(* CODESYS project TestProject.project

Project tree, tasks and I/O mapping:
  Jinan_Cherry_ARM_Cortex_VxWorks : Jinan Cherry-ARM Cortex-VxWorks, Jinan Cheery Electric Co., Ltd., version 3.5.11.20
    application Application
      libraries: CmpGlodonDemo, 1.0.0.0 (Glodon)
      task ConnectIOT (cyclic, interval t#2000ms, priority 1) calls DoConnectInternet
      task GetIOTData (cyclic, interval t#10000ms, priority 2) calls DoGetIOTData
      task UploadMachineData (cyclic, interval t#3000ms, priority 2) calls DoUploadIOTData
      task control_upload (cyclic, interval t#10000ms, priority 5) calls do_control_upload
      program DoConnectInternet [ST]
      program POU_1 [CFC]
      program DoGetIOTData [ST]
      global variables GVL_IOTData
      program DoUploadIOTData [ST]
      program do_control_upload [ST]
    SoftMotion General Axis Pool
*)

// Jinan_Cherry_ARM_Cortex_VxWorks/Application/GVL_IOTData
{attribute 'qualified_only'}
VAR_GLOBAL	
	//连网相关
	G_iotInitialized: BOOL;
	//测试开关
	G_uploadStartTask: BOOL;
	G_uploadUpdateTask: BOOL;
	G_uploadEndTask: BOOL;
	G_uploadMachineData: BOOL;
	
	G_nTaskCount: INT; //任务数量
	G_nCurTaskIndex: INT; //当前任务序号
	
    G_nBarLevel: INT; //钢筋级别
	G_rBarDiameter: REAL; //钢筋直径
	G_taskParams: ARRAY [1..10] OF TMP.OneSideParam; //	
	G_BarCount: INT; //加工钢筋根数
	G_TaskID: STRING; //任务ID
	
	G_nReturnValue: INT;
	
END_VAR

// Jinan_Cherry_ARM_Cortex_VxWorks/Application/DoConnectInternet
PROGRAM DoConnectInternet
VAR    
	fDoConnected: TMP.do_access_IOT;
END_VAR

//物联网心跳函数。保持2-3一次即可。优先级可以调低。
fDoConnected();

END_PROGRAM

// Jinan_Cherry_ARM_Cortex_VxWorks/Application/DoGetIOTData
//获取加工任务信息
//输入：加工任务序号
//输出：加工任务信息
//说明：该任务后续应作为任务触发（当点击获取任务使），而非循环事件
PROGRAM DoGetIOTData
VAR
	fGetTaskCount: TMP.get_task_count;
	fGetTaskData: TMP.get_task_data;
	G_nBarLevel: INT;
END_VAR

fGetTaskCount();
GVL_IOTData.G_nTaskCount := fGetTaskCount.nTaskCount;
GVL_IOTData.G_nCurTaskIndex := 0;
//获取一个任务的加工数据
fGetTaskData.nIndex := GVL_IOTData.G_nCurTaskIndex;
fGetTaskData();
//需要判断这个returnValue是否为0,0为获取成功
GVL_IOTData.G_nReturnValue := fGetTaskData.nReturnValue; 
GVL_IOTData.G_nBarLevel := fGetTaskData.nBarLevel;
GVL_IOTData.G_rBarDiameter := fGetTaskData.rBarDiameter;
GVL_IOTData.G_taskParams := fGetTaskData.taskParams;
GVL_IOTData.G_BarCount := fGetTaskData.nTaskCount;
GVL_IOTData.G_TaskID := fGetTaskData.taskID;

END_PROGRAM

// Jinan_Cherry_ARM_Cortex_VxWorks/Application/DoUploadIOTData
PROGRAM DoUploadIOTData
VAR
	fUploadMachineData: TMP.update_machine_data;
	fUploadStartTaskData: TMP.start_one_task;
	fUploadUpdateTaskData: TMP.update_one_task;
	fUploadEndTaskData: TMP.end_one_task;
END_VAR

//设备数据
IF GVL_IOTData.G_uploadMachineData THEN
	fUploadMachineData.iElectircFlow := 1000;
	fUploadMachineData.iOther := 'myTest';
	fUploadMachineData();
	//需要判断这个returnValue是否为0,0为上传成功
	GVL_IOTData.G_nReturnValue := fUploadMachineData.nReturnValue;
END_IF
//开始加工任务
IF GVL_IOTData.G_uploadStartTask THEN
	fUploadStartTaskData.nBarLevel := 3;
	fUploadStartTaskData.nParamCount := 2;
	fUploadStartTaskData.taskID := '123';
	fUploadStartTaskData.rBarDiameter := 8;
	fUploadStartTaskData.taskParams := GVL_IOTData.G_taskParams;
	fUploadStartTaskData();
	//需要判断这个returnValue是否为0,0为上传成功
	GVL_IOTData.G_nReturnValue := fUploadStartTaskData.nReturnValue;
END_IF
//结束加工任务
IF GVL_IOTData.G_uploadEndTask THEN
	fUploadEndTaskData.nCount := 20;
	fUploadEndTaskData.taskID := 'myTest';
	fUploadEndTaskData();
	//需要判断这个returnValue是否为0,0为上传成功
	GVL_IOTData.G_nReturnValue := fUploadEndTaskData.nReturnValue;
END_IF
//更新加工任务
IF GVL_IOTData.G_uploadUpdateTask THEN
	fUploadUpdateTaskData.nCount := 10;
	fUploadUpdateTaskData.taskID:= 'myTest';
	fUploadUpdateTaskData();
	//需要判断这个returnValue是否为0,0为上传成功
	GVL_IOTData.G_nReturnValue := fUploadUpdateTaskData.nReturnValue;
END_IF

END_PROGRAM

// Jinan_Cherry_ARM_Cortex_VxWorks/Application/do_control_upload
PROGRAM do_control_upload
VAR
END_VAR

GVL_IOTData.G_uploadStartTask := FALSE;
GVL_IOTData.G_uploadEndTask := FALSE;
GVL_IOTData.G_uploadMachineData := FALSE;
GVL_IOTData.G_uploadUpdateTask := TRUE;

END_PROGRAM

// Jinan_Cherry_ARM_Cortex_VxWorks/Application/POU_1
PROGRAM POU_1
VAR
	iTaskCount: INT;
END_VAR

END_PROGRAM
